FUNCTION F_GetROI : HRESULT
VAR_INPUT
	sFileName 			: 	REFERENCE TO STRING;
	stRoi				:	REFERENCE TO TcVnRectangle_UDINT;
	fThreshold			:	REFERENCE TO LREAL;
	bInvertImage		: 	REFERENCE TO BOOL;
	sPattern			:	REFERENCE TO STRING;
END_VAR
VAR
END_VAR

IF sFileName = 'OCR_01.png' THEN
	stRoi.nX := 86;
	stRoi.nY := 34;
	stRoi.nWidth := 263;
	stRoi.nHeight := 102;
	fThreshold := 150;
	bInvertImage := TRUE;
	sPattern := 'dd#dd#dd';
ELSIF sFileName = 'OCR_02.png' THEN
	stRoi.nX := 69;
	stRoi.nY := 40;
	stRoi.nWidth := 237;
	stRoi.nHeight := 80;
	fThreshold := 150;
	bInvertImage := TRUE;
	sPattern := 'dd#dd#dddd';
ELSIF sFileName = 'OCR_03.png' THEN
	stRoi.nX := 30;
	stRoi.nY := 40;
	stRoi.nWidth := 460;
	stRoi.nHeight := 110;
	fThreshold := 120;
	bInvertImage := TRUE;
	sPattern := 'udddudd###d';
ELSIF sFileName = 'OCR_04.png' THEN
	stRoi.nX := 131;
	stRoi.nY := 25;
	stRoi.nWidth := 243;
	stRoi.nHeight := 83;
	fThreshold := 75;
	bInvertImage := TRUE;
	sPattern := 'dd#dd#dddd';
ELSIF sFileName = 'OCR_05.png' THEN
	stRoi.nX := 129;
	stRoi.nY := 78;
	stRoi.nWidth := 257;
	stRoi.nHeight := 115;
	fThreshold := 150;
	bInvertImage := TRUE;
	sPattern := 'dd#dd#dd';
ELSIF sFileName = 'OCR_06.png' THEN
	stRoi.nX := 71;
	stRoi.nY := 50;
	stRoi.nWidth := 293;
	stRoi.nHeight := 101;
	fThreshold := 75;
	bInvertImage := TRUE;
	sPattern := 'dd#dd#dddd';
ELSIF sFileName = 'OCR_07.png' THEN
	stRoi.nX := 50;
	stRoi.nY := 120;
	stRoi.nWidth := 470;
	stRoi.nHeight := 110;
	fThreshold := 140;
	bInvertImage := FALSE;
	sPattern := 'udddudd###';
ELSIF sFileName = 'OCR_08.png' THEN
	stRoi.nX := 100;
	stRoi.nY := 83;
	stRoi.nWidth := 276;
	stRoi.nHeight := 108;
	fThreshold := 165;
	bInvertImage := TRUE;
	sPattern := 'dd#dd#dd';
ELSIF sFileName = 'OCR_09.png' THEN
	stRoi.nX := 90;
	stRoi.nY := 103;
	stRoi.nWidth := 284;
	stRoi.nHeight := 82; 
	fThreshold := 178;
	bInvertImage := TRUE;
	sPattern := 'dd#dd#dddd';
ELSIF sFileName = 'OCR_10.png' THEN
	stRoi.nX := 207;
	stRoi.nY := 4;
	stRoi.nWidth := 283;
	stRoi.nHeight := 104;
	fThreshold := 130;
	bInvertImage := TRUE;
	sPattern := 'dd#dd#dddd';
ELSIF sFileName = 'OCR_11.png' THEN
	stRoi.nX := 175;
	stRoi.nY := 245;
	stRoi.nWidth := 660;
	stRoi.nHeight := 115;
	fThreshold := 160;
	bInvertImage := TRUE;
	sPattern := 'uu#dddddddd';	
ELSIF sFileName = 'OCR_12.png' THEN 
	stRoi.nX := 74;
	stRoi.nY := 198;
	stRoi.nWidth := 248;
	stRoi.nHeight := 95;
	fThreshold := 130;
	bInvertImage := FALSE;
	sPattern := 'dd#dddd';
ELSIF sFileName = 'OCR_13.png' THEN
	stRoi.nX := 404;
	stRoi.nY := 2;
	stRoi.nWidth := 392;
	stRoi.nHeight := 159;
	fThreshold := 130;
	bInvertImage := FALSE;
	sPattern := 'dd#dd#dd';
ELSIF sFileName = 'OCR_14.png' THEN
	stRoi.nX := 260;
	stRoi.nY := 105;
	stRoi.nWidth := 340;
	stRoi.nHeight := 102;
	fThreshold := 160;
	bInvertImage := FALSE;
	sPattern := 'dd#dd#dddd';
ELSIF sFileName = 'OCR_15.png' THEN
	stRoi.nX := 250;
	stRoi.nY := 5;
	stRoi.nWidth := 560;
	stRoi.nHeight := 125;
	fThreshold := 160;
	bInvertImage := TRUE;
	sPattern := 'uddddd#dd#dd';
ELSIF sFileName = 'OCR_16.png' THEN
	stRoi.nX := 200;
	stRoi.nY := 0;
	stRoi.nWidth := 285;
	stRoi.nHeight := 70;
	fThreshold := 130;
	bInvertImage := FALSE;
	sPattern := 'dd#dd#dddd';
ELSIF sFileName = 'OCR_17.png' THEN
	stRoi.nX := 247;
	stRoi.nY := 83;
	stRoi.nWidth := 213;
	stRoi.nHeight := 94;
	fThreshold := 155;
	bInvertImage := FALSE;
	sPattern := 'dd#dddd';
ELSIF sFileName = 'OCR_18.png' THEN
	stRoi.nX := 25;
	stRoi.nY := 187;
	stRoi.nWidth := 330;
	stRoi.nHeight := 109;
	fThreshold := 100;
	bInvertImage := FALSE;
	sPattern := 'dd#dddd';
ELSIF sFileName = 'OCR_19.png' THEN
	stRoi.nX := 365;
	stRoi.nY := 70;
	stRoi.nWidth := 300;
	stRoi.nHeight := 95;
	fThreshold := 80;
	bInvertImage := TRUE;
	sPattern := 'uduuuud';
END_IF

END_FUNCTION

(* stored: Version 1.1.0.1, ProductVersion 3.1.4024.12
   POU F_GetROI: Id {32e039f3-9e63-4203-91dc-ee36d78793fb}, SpecialFunc None *)
